ABB RobotStudio station: Material Handeling (First Class).rsstn

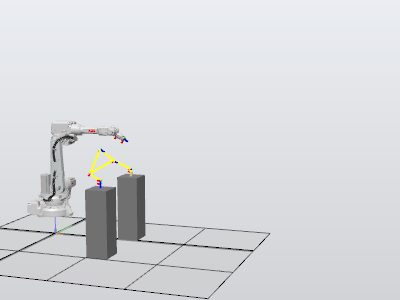
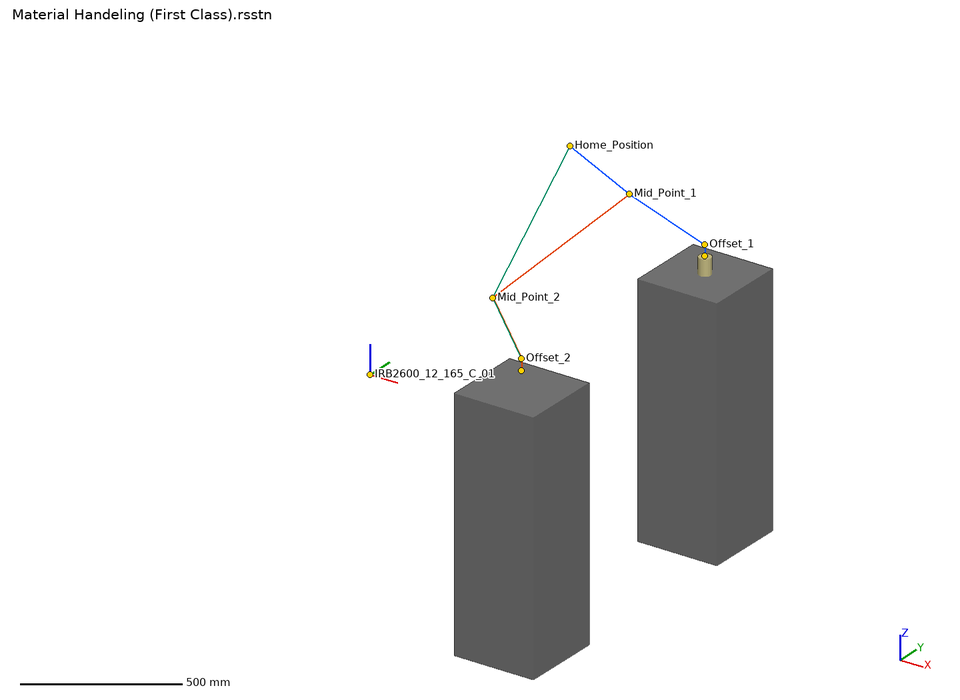
[picture v1: parts stored in the station drawn from their meshes, with robot base, taught points and paths (robot models come from the ABB library and are not in the file)]
Station Station (saved by RobotStudio 22.3.10141.1)
Controller Controller24, task T_ROB1: task frame (RAPID world) sits at (0, 0, 290) mm in the station
Controller Controller24
  mechanical unit ROB_1: IRB2600_12_165_C_01, 6 joints, base frame (0, 0, 0) mm
Layout (positions relative to the parent item):
  - IRB2600_12_165_C_01 [mechanism, from %ABB.RobotStudio.Models.IRB2600%\IRB2600_12_165_C_01.rslib] at (0, 0, 290) mm; joint values [0, 0, 0, 0, 0.5236, 0] (rad or m)
  - SmartComponent_1 [smart component]
      signals: DI di_attach, DO Do_led
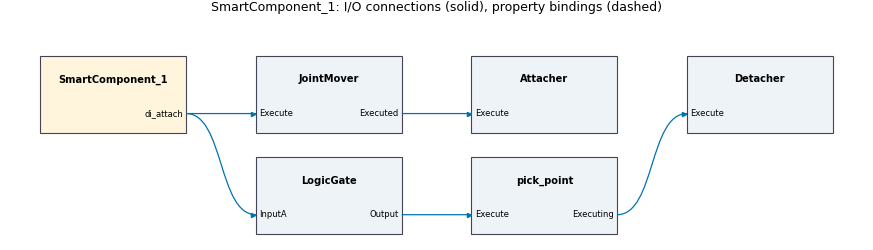
      connections:
        SmartComponent_1.di_attach -> JointMover.Execute
        SmartComponent_1.di_attach -> LogicGate.InputA
        LogicGate.Output -> pick_point.Execute
        pick_point.Executing -> Detacher.Execute
        JointMover.Executed -> Attacher.Execute
    - Smart_Gripper_Servo_Fingers [mechanism, from Tools\ABB_Smart_Gripper_Servo_Fingers.rslib] at (1018.61, 0, 1507.5) mm, rotated rx 180 ry 60 rz 180 deg; joint values [0.025] (rad or m)
    - Detacher [smart component, from Components\Detacher.rslib]
        properties: Child=Object_1; KeepPosition=true
    - Attacher [smart component, from Components\Attacher.rslib]
        properties: Parent=Smart_Gripper_Servo_Fingers; Flange=0; Child=Object_1; Mount=false; Offset=[0 0 0]; Orientation=[0 0 0]
    - LogicGate [smart component, from Components\LogicGate.rslib]
        properties: Operator=NOT; Delay=0
    - JointMover [smart component, from Components\JointMover.rslib]
        properties: Mechanism=Smart_Gripper_Servo_Fingers; Relative=false; Duration=0; J1=0.0225
    - pick_point [smart component, from Components\JointMover.rslib]
        properties: Mechanism=Smart_Gripper_Servo_Fingers; Relative=false; Duration=0; J1=0.025
  - Piller_1 [part] at (1003.05, -982.86, 0) mm, size 300 x 300 x 900 mm
  - Piller_2 [part] at (1006.06, 0, 0) mm, size 300 x 300 x 900 mm
  - Object_2 [part] at (1153.05, -832.86, 900) mm, size 45 x 44.7 x 60 mm
  - Object_1 [part] at (1156.06, 150, 900) mm, size 45 x 44.7 x 60 mm
Attachment: Smart_Gripper_Servo_Fingers is attached to IRB2600_12_165_C_01 / Link6
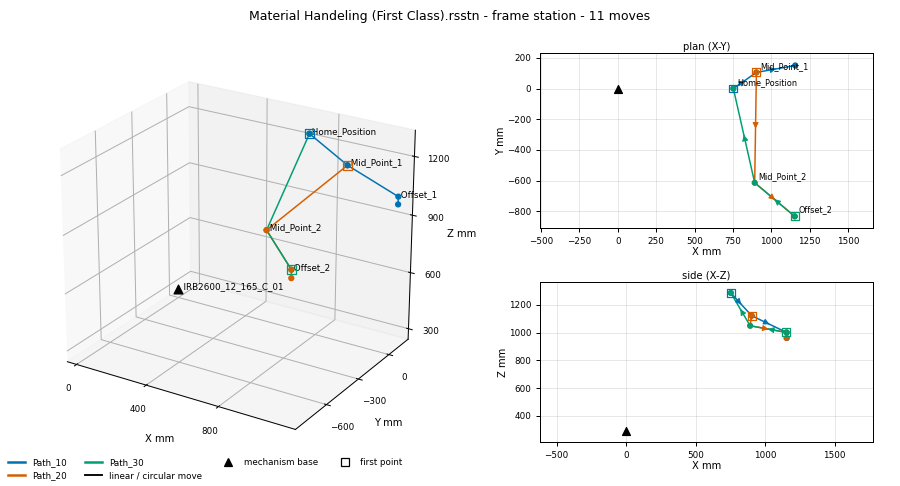
[picture p0: tool path of Material Handeling (First Class).rsstn in frame station, 11 of 11 moves have a stored position in this frame; points joined in program order, loops and branches not executed]
Targets, tools, work objects and paths stored in the station, written as RAPID:
! task T_ROB1
MODULE CalibData
  PERS tooldata Servo:=[TRUE,[[0,0,114.2],[1,0,0,0]],[0.215,[8.7,12.3,49.2],[1,0,0,0],0.00021,0.00024,0.00009]];
ENDMODULE

! task T_ROB1
MODULE Module1
  CONST robtarget Home_Position:=[[753.132200933,0,994.852758437],[0.50000002,0,0.866025392,0],[0,0,0,0],[9E+09,9E+09,9E+09,9E+09,9E+09,9E+09]];
  CONST robtarget Mid_Point_1:=[[903.209742311,105.069431959,830.875617836],[0.500000145,0.000000004,0.86602532,-0.000000017],[0,-1,0,0],[9E+09,9E+09,9E+09,9E+09,9E+09,9E+09]];
  CONST robtarget Pick_Point_1:=[[1156.061989137,150.000090514,669.999813984],[0.012183432,-0.000000074,-0.999925779,0],[0,0,0,0],[9E+09,9E+09,9E+09,9E+09,9E+09,9E+09]];
  CONST robtarget Offset_1:=[[1156.061985284,150.000089711,709.819047482],[0.012183436,-0.000000081,-0.999925779,0.000000002],[0,0,0,0],[9E+09,9E+09,9E+09,9E+09,9E+09,9E+09]];
  CONST robtarget Mid_Point_2:=[[892.035163981,-613.883222862,758.684530835],[0.500000113,-0.000000058,0.866025338,-0.000000039],[-1,0,-2,0],[9E+09,9E+09,9E+09,9E+09,9E+09,9E+09]];
  CONST robtarget Place_Point:=[[1153.053032566,-832.860395776,669.999699725],[0.008081702,-0.000000076,0.999967343,0.00000004],[-1,0,-1,0],[9E+09,9E+09,9E+09,9E+09,9E+09,9E+09]];
  CONST robtarget Offset_2:=[[1153.053040524,-832.860401365,710.754924787],[0.008081745,-0.000000069,0.999967342,0.00000001],[-1,0,-1,0],[9E+09,9E+09,9E+09,9E+09,9E+09,9E+09]];
  PROC Path_10()
    MoveL Home_Position,v1000,z100,Servo\WObj:=wobj0;
    MoveL Mid_Point_1,v1000,z100,Servo\WObj:=wobj0;
    MoveL Offset_1,v1000,z100,Servo\WObj:=wobj0;
    MoveL Pick_Point_1,v1000,z100,Servo\WObj:=wobj0;
  ENDPROC
  PROC Path_20()
    MoveL Mid_Point_1,v1000,z100,Servo\WObj:=wobj0;
    MoveL Mid_Point_2,v1000,z100,Servo\WObj:=wobj0;
    MoveL Offset_2,v1000,z100,Servo\WObj:=wobj0;
    MoveL Place_Point,v1000,z100,Servo\WObj:=wobj0;
  ENDPROC
  PROC Path_30()
    MoveL Offset_2,v1000,z100,Servo\WObj:=wobj0;
    MoveL Mid_Point_2,v1000,z100,Servo\WObj:=wobj0;
    MoveL Home_Position,v1000,z100,Servo\WObj:=wobj0;
  ENDPROC
ENDMODULE

